{attribute 'GeneratedUsingTerminal: EL2912-0000-0016'}
{attribute addProperty BoxType "EL2912-0000-0016"}
{attribute addProperty Id "FSOEAT %I*FSOE_046F804E7"}
{attribute addProperty CRC "2476392253"}
{attribute addProperty Size "7"}
TYPE FSoE_Inputs_939ABF3D :
STRUCT
	{attribute addProperty Name "FSOE"}
	FSOE AT %I* : FSOE_046F804E;
END_STRUCT
END_TYPE

(* stored: Version 1.2.0.0, ProductVersion 3.1.4024.9
   DUT FSoE_Inputs_939ABF3D: Id {c3cd9993-835e-4052-965f-e63a71ca87e8} *)
